(* IEC 61131-3 sources: eCockpitGit/test_project/src/%F%00 Library/%F%Common Functions/%F%Dynamic Array/%F%Dynamic Array Orderly (Obsolete), 6 files *)

(* ---- %POU%FU_dynamicArrayTransfer.st ---- *)
//This allocates the needed size for the array
// |**Version**|**Author**| **Date** |**Changes**
// | 1         | NSN      | 24-11-20 | Creation
FUNCTION FU_dynamicArrayTransfer : BOOL
VAR_INPUT
	oldArray		:POINTER TO BYTE;
	newArray		:POINTER TO BYTE;
	oldSize			:WORD;
	newSize			:WORD;
END_VAR
VAR
	smallest		:DINT;
	i				:DINT;
END_VAR
(*%!%__DELIMITER__%!%*)
smallest			:=		MIN(oldSize,newSize);
FOR i := 1 TO smallest DO
	newArray^		:=		oldArray^;
	newArray		:=		newArray + 1;
	oldArray		:=		oldArray + 1;
END_FOR

(* ---- %POU%FU_DynPointArrayIncSize.st ---- *)
//This increases the size of a dynamic array of pointers
//Returns OutOfDynamicMemory when memory allocation fails
// |**Version**|**Author**| **Date** |**Changes**
// | 1         | NSN      | 16-12-20 | Creation
FUNCTION FU_DynPointArrayIncSize:SLMResult
VAR_IN_OUT
	workingArray		:POINTER TO ARRAY[0..999] OF POINTER TO BYTE;	//Array
END_VAR
VAR_INPUT
	incrementAmount		:WORD;	//How much to increase the size of the array by at a time, keep this value the same all the time
END_VAR
VAR_OUTPUT
	arraySize			:WORD;	//Size of new array
END_VAR
VAR
	arrayBuffer			:POINTER TO ARRAY[0..999] OF POINTER TO BYTE;	//
	arrayDelete			:POINTER TO ARRAY[0..999] OF POINTER TO BYTE;	//Buffer for deallocating buffer memory
	arraySizeNew		:WORD;	//Size of new array
	i					:WORD;
END_VAR
(*%!%__DELIMITER__%!%*)
//Size of old memory is retrieved
arraySize								:=		TO_WORD(FU_getBlockSizeFromPointer(pData:=workingArray) / 4);
//If there is no space, the memory manager is queried for a new bigger buffer
arraySizeNew							:=		arraySize + incrementAmount;
arrayBuffer								:=		__NEW(POINTER TO BYTE,arraySizeNew);
//If the memory manager fails, the registerering fails
IF arrayBuffer = 0 THEN
	FU_DynPointArrayIncSize.code		:=		ERCodes.DynPointArrayIncSize;
	FU_DynPointArrayIncSize.reason		:=		GTErrors.EoutOfDynamicMemory;
	FU_DynPointArrayIncSize.success		:=		FALSE;
	RETURN;
END_IF
//The contens of the old buffer is copied to the new buffer
IF arraySize > 0 THEN
	FOR i := 0 TO arraySize - 1 DO
		arrayBuffer^[i]					:=		workingArray^[i];
	END_FOR
END_IF
//Old memory is stored for deletion
arrayDelete								:=		workingArray;
//Old buffer is overwritten with new buffer
workingArray							:=		arrayBuffer;
arraySize								:=		arraySize + incrementAmount;
//The old buffer is deregistered
FU_SafeDelete(pMem:=arrayDelete);

(* ---- %POU%FU_DynPointArrayOrderAdd.st ---- *)
//This adds a pointer to a dynamic pointer array, if the array is full it increments the size of the array
//It is orderly meaning that all the stored ids are one after the other
//This ensures that a process can loop through all entries without checking for null pointers and only until the array amount value is reached
//Returns OutOfDynamicMemory when memory allocation fails
//Returns AlreadyInRegistry if pointer is already in array
//Returns VarsWrong if invalid pointer is given
// |**Version**|**Author**| **Date** |**Changes**
// | 1         | NSN      | 16-12-20 | Creation
FUNCTION FU_DynPointArrayOrderAdd:SLMResult
VAR_IN_OUT
	arrayAmount			:WORD;	//Amount in array
	workingArray		:POINTER TO ARRAY[0..999] OF POINTER TO BYTE;	//Array
END_VAR
VAR_INPUT
	addPoint			:POINTER TO BYTE;	//The pointer to add
	incrementAmount		:WORD;	//How much to increase the size of the array by at a time, keep this value the same all the time
END_VAR
VAR
	arraySize			:DWORD;
END_VAR
(*%!%__DELIMITER__%!%*)
//Check for valid pointer
IF addPoint = 0 THEN
	FU_DynPointArrayOrderAdd.code		:=		ERCodes.DynPointArrayOrderAdd;
	FU_DynPointArrayOrderAdd.reason		:=		GTErrors.EinvalidPointer;
	FU_DynPointArrayOrderAdd.success	:=		FALSE;
	RETURN;
END_IF
//Checks if pointer is already in array
IF FU_DynPointArrayOrderCheckDupe(arrayAmount:=arrayAmount,workingArray:=workingArray,checkPoint:=addPoint) THEN
	FU_DynPointArrayOrderAdd.code		:=		ERCodes.DynPointArrayOrderAdd;
	FU_DynPointArrayOrderAdd.reason		:=		GTErrors.EpointerAlreadyRegistered;
	FU_DynPointArrayOrderAdd.success	:=		FALSE;
	RETURN;
END_IF
//Size of memory is retrived
arraySize						:=		FU_getBlockSizeFromPointer(pData:=workingArray) / 4;

//This checks if there is space left in the managers buffer
IF arrayAmount = arraySize THEN
	FU_DynPointArrayOrderAdd	:=		FU_DynPointArrayIncSize(workingArray:=workingArray,incrementAmount:=incrementAmount);
	IF NOT(FU_DynPointArrayOrderAdd.success) THEN
		RETURN;
	END_IF
END_IF
workingArray^[arrayAmount]		:=		addPoint;
arrayAmount						:=		arrayAmount + 1;

(* ---- %POU%FU_DynPointArrayOrderCheckDupe.st ---- *)
//This checks if a pointer is inside a dynamic pointer array
//Returns true if a duplicate is found
// |**Version**|**Author**| **Date** |**Changes**
// | 1         | NSN      | 16-12-20 | Creation
FUNCTION FU_DynPointArrayOrderCheckDupe:BOOL
VAR_IN_OUT
	arrayAmount			:WORD;	//Amount in array
	workingArray		:POINTER TO ARRAY[0..999] OF POINTER TO BYTE;	//Array
END_VAR
VAR_INPUT
	checkPoint			:POINTER TO BYTE;	//The pointer to remove from the array
END_VAR
VAR
	i					:WORD;
END_VAR
(*%!%__DELIMITER__%!%*)
//Check for valid pointer
IF checkPoint = 0 THEN
	RETURN;
END_IF
IF arrayAmount > 0 THEN
	FOR i := 0 TO arrayAmount - 1 DO
		IF checkPoint = workingArray^[i] THEN
			FU_DynPointArrayOrderCheckDupe	:=		TRUE;
			RETURN;
		END_IF
	END_FOR
END_IF

(* ---- %POU%FU_DynPointArrayOrderRemove.st ---- *)
//This removes a pointer from a dynamic pointer array
//It also moves all the ids after it to close the gap left
// |**Version**|**Author**| **Date** |**Changes**
// | 1         | NSN      | 16-12-20 | Creation
//Returns true if the pointer was found in the array
FUNCTION FU_DynPointArrayOrderRemove:BOOL
VAR_IN_OUT
	arrayAmount			:WORD;	//Amount in array
	workingArray		:POINTER TO ARRAY[0..999] OF POINTER TO BYTE;	//Array
END_VAR
VAR_INPUT
	removePoint			:POINTER TO BYTE;	//The pointer to remove from the array
END_VAR
VAR_OUTPUT
	index				:WORD;			//Index of removed array pointer
END_VAR
VAR
	amountBuff			:WORD;
	offSet				:BYTE;
	i					:WORD;
END_VAR
(*%!%__DELIMITER__%!%*)
//Check for valid pointer
IF removePoint = 0 THEN
	RETURN;
END_IF
amountBuff										:=		arrayAmount;
IF arrayAmount > 0 THEN
	IF arrayAmount > 1 THEN
		FOR i := 0 TO amountBuff - offSet - 1 DO
			IF removePoint = workingArray^[i] THEN
				FU_DynPointArrayOrderRemove		:=		TRUE;
				arrayAmount						:=		arrayAmount - 1;
				offSet							:=		offSet + 1;
				index							:=		i;
			END_IF
			IF FU_DynPointArrayOrderRemove AND i < arrayAmount THEN
				workingArray^[i]				:=		workingArray^[i + offSet];
			END_IF
		END_FOR
	ELSE
		IF removePoint = workingArray^[0] THEN
			FU_DynPointArrayOrderRemove			:=		TRUE;
			arrayAmount							:=		arrayAmount - 1;
		END_IF
	END_IF
	IF FU_DynPointArrayOrderRemove THEN
		workingArray^[i]						:=		0;
	END_IF
END_IF

(* ---- %POU%FU_getBlockSizeFromPointer.st ---- *)
//Finds the block header from a codesys dynamic memory block
// |**Version**|**Author**| **Date** |**Changes**
// | 1         | NSN      | 16-12-20 | Creation
FUNCTION FU_getBlockSizeFromPointer : DWORD
VAR_INPUT
	pData		:POINTER TO BYTE;
END_VAR
var
	pHeader		:POINTER TO CMM.LMMBlock := pData - 12;
END_VAR
(*%!%__DELIMITER__%!%*)
IF pData <> 0 THEN
	FU_getBlockSizeFromPointer			:=		pHeader^.dwSize - 16;
ELSE
	FU_getBlockSizeFromPointer			:=		0;
END_IF
